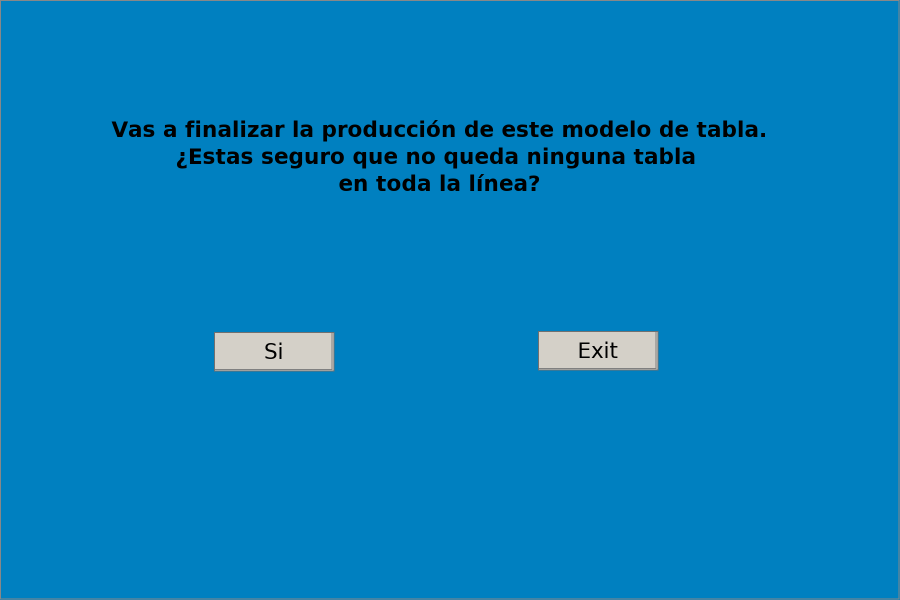
VISUALIZATION V_Emergente_Fin_Produccion  // 900x600
    Button (214,332 120x39), "Si"
        tap FuncParoNodoCorteH4Remote1.FunGeneCortHum4.P_FinProduccion p3779583253=TRUE
        OnMouseClick: change screen: Modelo_Tabla
        OnMouseClick: CloseDialog Dialog=V_Emergente_Fin_Produccion, Result=OK, NumpadKeypadSet=True
    Button (538,331 120x39), "Exit"
        OnMouseClick: CloseDialog Dialog=V_Emergente_Fin_Produccion, Result=OK, NumpadKeypadSet=True
    Label (113,67 653x179), "Vas a finalizar la producción de este modelo de tabla. ¿Estas seguro que no queda ninguna tabla en toda la línea?"
END_VISUALIZATION

(* stored: Version 1.1.0.1, ProductVersion 3.1.4024.12
   Visu V_Emergente_Fin_Produccion: Id {86e0ce7c-4ab9-4540-bcf4-39651436cbcb} *)
